Yaskawa INFORM job: aruba_cylinder_program.JBI

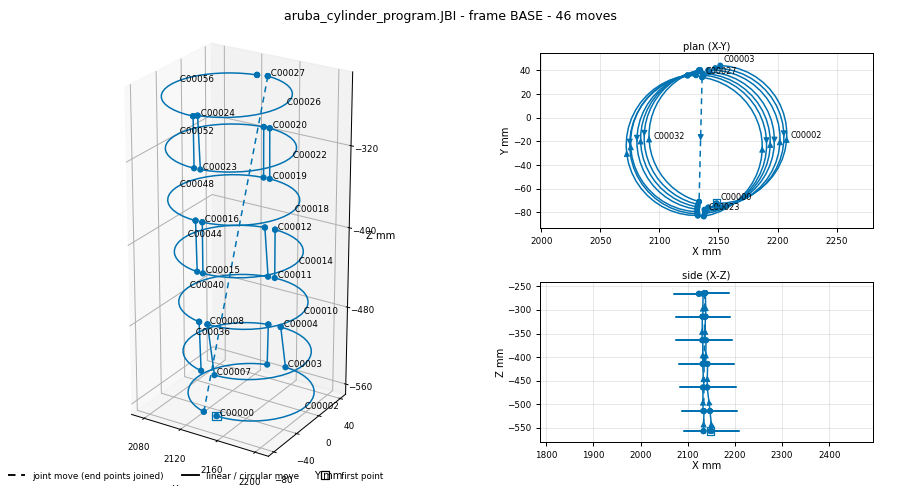
[picture p0: tool path of aruba_cylinder_program.JBI in frame BASE, 46 of 66 moves have a stored position in this frame; points joined in program order, loops and branches not executed]
/JOB
//NAME aruba_cylinder_program
//POS
///NPOS 60,0,60,0,0,0
///TOOL 0
///POSTYPE BASE
///RECTAN
///RCONF 0,0,0,0,0,0,0,0,0,0,0,0,0,0,0,0,0,0,0,0,0,0,0,0
C00000=2148.360000,-72.440900,-556.605500,90.000000,-90.000000,5.000000
C00001=2148.360000,-72.440900,-556.605500,90.000000,-90.000000,5.000000
C00002=2207.600000,-19.912500,-556.605500,175.000000,-89.999999,5.000000
C00003=2151.520000,44.207200,-556.605500,-90.000000,-90.000000,5.000000
C00004=2147.280000,41.889600,-514.228000,-90.000000,-90.000000,5.000000
C00005=2147.280000,41.889600,-514.228000,-90.000000,-90.000000,5.000000
C00006=2205.380000,-13.272300,-514.228000,175.000000,-89.999999,5.000000
C00007=2147.470000,-74.286700,-514.228000,90.000000,-90.000000,5.000000
C00008=2141.370000,-75.913100,-464.228000,90.000000,-90.000000,5.000000
C00009=2141.370000,-75.913100,-464.228000,90.000000,-90.000000,5.000000
C00010=2202.020000,-14.019100,-464.228000,175.000000,-89.999999,5.000000
C00011=2141.260000,40.308100,-464.228000,-90.000000,-90.000000,5.000000
C00012=2142.190000,38.821400,-414.228000,-90.000000,-90.000000,5.000000
C00013=2142.190000,38.821400,-414.228000,-90.000000,-90.000000,5.000000
C00014=2197.340000,-16.966900,-414.228000,175.000000,-89.999999,5.000000
C00015=2138.110000,-77.733800,-414.228000,90.000000,-90.000000,5.000000
C00016=2138.910000,-79.347000,-364.228000,90.000000,-90.000000,5.000000
C00017=2138.910000,-79.347000,-364.228000,90.000000,-90.000000,5.000000
C00018=2193.810000,-17.908900,-364.228000,175.000000,-89.999999,5.000000
C00019=2136.880000,37.419400,-364.228000,-90.000000,-90.000000,5.000000
C00020=2137.420000,36.079800,-314.228000,-90.000000,-90.000000,5.000000
C00021=2137.420000,36.079800,-314.228000,-90.000000,-90.000000,5.000000
C00022=2190.570000,-17.264600,-314.228000,175.000000,-89.999999,5.000000
C00023=2138.360000,-80.950100,-314.228000,90.000000,-90.000000,5.000000
C00024=2137.560000,-83.409000,-263.917500,90.000000,-90.000000,5.000000
C00025=2137.560000,-83.409000,-263.917500,90.000000,-90.000000,5.000000
C00026=2187.060000,-22.020800,-263.917500,175.000000,-89.999999,5.000000
C00027=2136.170000,34.271600,-263.917500,-90.000000,-90.000000,5.000000
C00028=2136.170000,34.271600,-263.917500,-90.000000,-90.000000,5.000000
C00029=2136.170000,34.271600,-263.917500,-90.000000,-90.000000,5.000000
C00030=2133.610000,-70.976200,-557.001500,90.000000,-90.000000,5.000000
C00031=2133.610000,-70.976200,-557.001500,90.000000,-90.000000,5.000000
C00032=2091.520000,-21.465100,-557.001500,5.000000,-89.999999,5.000000
C00033=2133.490000,40.392400,-557.001500,-90.000000,-90.000000,5.000000
C00034=2134.550000,40.359700,-514.228000,-90.000000,-90.000000,5.000000
C00035=2134.550000,40.359700,-514.228000,-90.000000,-90.000000,5.000000
C00036=2087.100000,-16.815500,-514.228000,5.000000,-89.999999,5.000000
C00037=2132.560000,-73.356900,-514.228000,90.000000,-90.000000,5.000000
C00038=2132.220000,-75.502800,-464.228000,90.000000,-90.000000,5.000000
C00039=2132.220000,-75.502800,-464.228000,90.000000,-90.000000,5.000000
C00040=2084.190000,-21.826900,-464.228000,5.000000,-89.999999,5.000000
C00041=2134.500000,39.433800,-464.228000,-90.000000,-90.000000,5.000000
C00042=2131.580000,38.031500,-414.228000,-90.000000,-90.000000,5.000000
C00043=2131.580000,38.031500,-414.228000,-90.000000,-90.000000,5.000000
C00044=2080.940000,-19.750400,-414.228000,5.000000,-89.999999,5.000000
C00045=2131.940000,-77.487800,-414.228000,90.000000,-90.000000,5.000000
C00046=2132.030000,-79.560300,-364.228000,90.000000,-90.000000,5.000000
C00047=2132.030000,-79.560300,-364.228000,90.000000,-90.000000,5.000000
C00048=2075.660000,-23.565200,-364.228000,5.000000,-89.999999,5.000000
C00049=2130.560000,37.000700,-364.228000,-90.000000,-90.000000,5.000000
C00050=2131.060000,36.010800,-314.228000,-90.000000,-90.000000,5.000000
C00051=2131.060000,36.010800,-314.228000,-90.000000,-90.000000,5.000000
C00052=2074.880000,-21.424500,-314.228000,5.000000,-89.999999,5.000000
C00053=2132.130000,-81.339400,-314.228000,90.000000,-90.000000,5.000000
C00054=2132.550000,-82.733700,-265.632500,90.000000,-90.000000,5.000000
C00055=2132.550000,-82.733700,-265.632500,90.000000,-90.000000,5.000000
C00056=2072.250000,-17.091600,-265.632500,5.000000,-89.999999,5.000000
C00057=2123.860000,35.842200,-265.632500,-90.000000,-90.000000,5.000000
C00058=2123.860000,35.842200,-265.632500,-90.000000,-90.000000,5.000000
C00059=2123.860000,35.842200,-265.632500,-90.000000,-90.000000,5.000000
///POSTYPE PULSE
///PULSE
EC00000=0
EC00001=0
EC00002=0
EC00003=0
EC00004=0
EC00005=0
EC00006=0
EC00007=0
EC00008=0
EC00009=0
EC00010=0
EC00011=0
EC00012=0
EC00013=0
EC00014=0
EC00015=0
EC00016=0
EC00017=0
EC00018=0
EC00019=0
EC00020=0
EC00021=0
EC00022=0
EC00023=0
EC00024=0
EC00025=0
EC00026=0
EC00027=0
EC00028=92160
EC00029=184320
EC00030=184320
EC00031=184320
EC00032=184320
EC00033=184320
EC00034=184320
EC00035=184320
EC00036=184320
EC00037=184320
EC00038=184320
EC00039=184320
EC00040=184320
EC00041=184320
EC00042=184320
EC00043=184320
EC00044=184320
EC00045=184320
EC00046=184320
EC00047=184320
EC00048=184320
EC00049=184320
EC00050=184320
EC00051=184320
EC00052=184320
EC00053=184320
EC00054=184320
EC00055=184320
EC00056=184320
EC00057=184320
EC00058=276480
EC00059=368640
//INST
///DATE 2023/05/18 10:31
///ATTR SC,RW,RJ
////FRAME BASE
///GROUP1 RB1,ST1
NOP
MOVJ P009 EX000 VJ=15.00
MOVJ P009 VJ=15.00
MOVJ C00000 EC00000 VJ=15.0
CALL JOB:SPYON
MOVC C00001 EC00001 V=150.0
MOVC C00002 EC00002 V=150.0
MOVC C00003 EC00003 V=150.0
MOVL C00004 EC00004 V=150.0
MOVC C00005 EC00005 V=150.0
MOVC C00006 EC00006 V=150.0
MOVC C00007 EC00007 V=150.0
MOVL C00008 EC00008 V=150.0
MOVC C00009 EC00009 V=150.0
MOVC C00010 EC00010 V=150.0
MOVC C00011 EC00011 V=150.0
MOVL C00012 EC00012 V=150.0
MOVC C00013 EC00013 V=150.0
MOVC C00014 EC00014 V=150.0
MOVC C00015 EC00015 V=150.0
MOVL C00016 EC00016 V=150.0
MOVC C00017 EC00017 V=150.0
MOVC C00018 EC00018 V=150.0
MOVC C00019 EC00019 V=150.0
MOVL C00020 EC00020 V=150.0
MOVC C00021 EC00021 V=150.0
MOVC C00022 EC00022 V=150.0
MOVC C00023 EC00023 V=150.0
MOVL C00024 EC00024 V=150.0
MOVC C00025 EC00025 V=150.0
MOVC C00026 EC00026 V=150.0
MOVC C00027 EC00027 V=150.0
CALL JOB:SPYOF
MOVJ P009 VJ=15.00
MOVL C00028 EC00028 V=150.0
MOVJ P009 VJ=15.00
MOVL C00029 EC00029 V=150.0
MOVJ C00030 EC00030 VJ=15.0
CALL JOB:SPYON
MOVC C00031 EC00031 V=150.0
MOVC C00032 EC00032 V=150.0
MOVC C00033 EC00033 V=150.0
MOVL C00034 EC00034 V=150.0
MOVC C00035 EC00035 V=150.0
MOVC C00036 EC00036 V=150.0
MOVC C00037 EC00037 V=150.0
MOVL C00038 EC00038 V=150.0
MOVC C00039 EC00039 V=150.0
MOVC C00040 EC00040 V=150.0
MOVC C00041 EC00041 V=150.0
MOVL C00042 EC00042 V=150.0
MOVC C00043 EC00043 V=150.0
MOVC C00044 EC00044 V=150.0
MOVC C00045 EC00045 V=150.0
MOVL C00046 EC00046 V=150.0
MOVC C00047 EC00047 V=150.0
MOVC C00048 EC00048 V=150.0
MOVC C00049 EC00049 V=150.0
MOVL C00050 EC00050 V=150.0
MOVC C00051 EC00051 V=150.0
MOVC C00052 EC00052 V=150.0
MOVC C00053 EC00053 V=150.0
MOVL C00054 EC00054 V=150.0
MOVC C00055 EC00055 V=150.0
MOVC C00056 EC00056 V=150.0
MOVC C00057 EC00057 V=150.0
CALL JOB:SPYOF
MOVJ P009 VJ=15.00
MOVL C00058 EC00058 V=150.0
MOVJ P009 VJ=15.00
MOVL C00059 EC00059 V=150.0
END
